FUNCTION_BLOCK E_MUX_2 (* Service Interface Function Block Type *)
  (* Standard: 61499-2 *)
  (* Version 0.0, 2008-07-10, 4DIAC-IDE, 4DIAC-Consortium *)
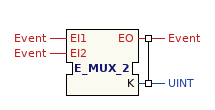
  EVENT_INPUT
    EI1; (* Mux in event *)
    EI2; (* Mux in event *)
  END_EVENT
  EVENT_OUTPUT
    EO WITH K; (* Mux output event *)
  END_EVENT
  VAR_OUTPUT
    K : UINT; (* Mux event index *)
  END_VAR
  (* Service APPLICATION/RESOURCE: Service Interface Function Block Type *)
END_FUNCTION_BLOCK
